TYPE System_Senser :
STRUCT
END_STRUCT
END_TYPE

(* stored: Version 1.1.0.1, ProductVersion 3.1.4024.9
   DUT System_Senser: Id {e0939ac8-e2d5-45ba-bf9c-8b468b16242c} *)
